FUNCTION TryConvert_TOD_TO_LREAL : BOOL
VAR_INPUT
	in : TOD;
	out : REFERENCE TO LREAL;
END_VAR

out := TOD_TO_LREAL(in);
TryConvert_TOD_TO_LREAL := TRUE;

END_FUNCTION

(* stored: Version 1.1.0.1, ProductVersion 3.1.4024.12
   POU TryConvert_TOD_TO_LREAL: Id {6c049ce6-df49-4217-933d-a7a54ee70bcf}, SpecialFunc None *)
